TYPE E_MoMa_2ndHierarchy_Implementation :
(
	Decision,
	MovingTM,
	MovingLD,
	VisionTask
)UDINT;
END_TYPE

(* stored: Version 1.1.0.1, ProductVersion 3.1.4024.11
   DUT E_MoMa_2ndHierarchy_Implementation: Id {a2eaedf1-925b-467d-9919-6eefe195c1d8} *)
